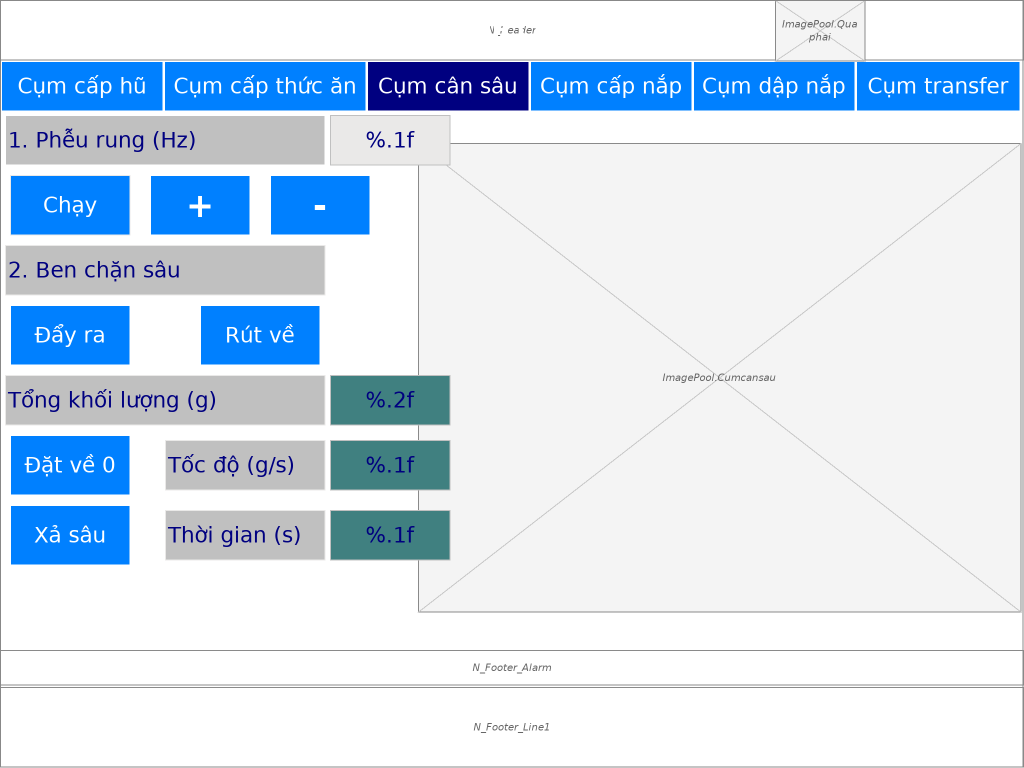
VISUALIZATION N_WormWeight1  // 1024x768
    Image (418,143 603x469), image: ImagePool.Cumcansau
    Rectangle (10,175 120x60), "Dừng", invisible if: not PR_Line01.bMotor_vibrating_funnel, input disabled if: not PR_Line01.bMotor_vibrating_funnel
        OnMouseDown: execute { PR_Line01.bMotor_vibrating_funnel := FALSE; PR_Line01.bxa := FALSE; }
    Rectangle (10,175 120x60), "Chạy", invisible if: PR_Line01.bMotor_vibrating_funnel, input disabled if: PR_Line01.bMotor_vibrating_funnel
        OnMouseDown: execute { PR_Line01.bMotor_vibrating_funnel := TRUE; PR_Line01.bxa := FALSE; }
    Rectangle (10,305 120x60), "Đẩy ra", colour toggle: PR_Line01.bCylinder_Block_Worm_Extend
        OnMouseDown: execute {
            PR_Line01.bCylinder_Block_Worm_Extend := TRUE;
            PR_Line01.bCylinder_Block_Worm_Retract := FALSE;
            PR_Line01.bxa := FALSE;
        }
    Rectangle (200,305 120x60), "Rút về", colour toggle: PR_Line01.bCylinder_Block_Worm_Retract
        OnMouseDown: execute {
            PR_Line01.bCylinder_Block_Worm_Retract := TRUE;
            PR_Line01.bCylinder_Block_Worm_Extend := FALSE;
            PR_Line01.bxa := FALSE;
        }
    Frame (0,687 1024x80)
        shows N_Footer_Line1()
    Frame (0,0 1024x60)
        shows N_Header()
    Textfield (353,5 400x50), "MÀN HÌNH CHẠY TAY LINE 1"
    Rectangle (5,115 320x50), "1. Phễu rung (Hz)"
    Rectangle (5,245 320x50), "2. Ben chặn sâu"
    Rectangle (1,61 162x50), "Cụm cấp hũ"
        OnMouseClick: change screen: N_JarSupply1
    Rectangle (164,61 202x50), "Cụm cấp thức ăn"
        OnMouseClick: change screen: N_FoodSupply1
    Rectangle (367,61 162x50), "Cụm cân sâu"
        OnMouseClick: change screen: N_WormWeight1
    Rectangle (530,61 162x50), "Cụm cấp nắp"
        OnMouseClick: change screen: N_LidSupply1
    Rectangle (693,61 162x50), "Cụm dập nắp"
        OnMouseClick: change screen: N_LidPressing1
    Rectangle (856,61 164x50), "Cụm transfer"
        OnMouseClick: change screen: N_Tranfer1
    Rectangle (330,115 120x50), "%.1f", text variable: PR_Line01.fb_WormWeight.fSpeed_vibrating_funnel_Manual
        OnMouseDown: write PR_Line01.fb_WormWeight.fSpeed_vibrating_funnel_Manual via VisuDialogs.Numpad
        OnMouseDown: execute { PR_Line01.bxa := FALSE; }
    Rectangle (5,375 320x50), "Tổng khối lượng (g)"
    Rectangle (150,175 100x60), "+", colour toggle: PR_Line01.bUp_vibrating_funnel
        OnMouseDown: execute { PR_Line01.bUp_vibrating_funnel := TRUE; PR_Line01.bxa := FALSE; }
    Rectangle (270,175 100x60), "-", colour toggle: PR_Line01.bDown_vibrating_funnel
        OnMouseDown: execute { PR_Line01.bDown_vibrating_funnel := TRUE; PR_Line01.bxa := FALSE; }
    Rectangle (330,375 120x50), "%.2f", text variable: PR_Line01.fb_WormWeight.fWeight_Worm
    Rectangle (10,435 120x60), "Đặt về 0"
        tap PR_Line01.bZero_Loadcell_Worm
        OnMouseDown: execute { PR_Line01.bxa := FALSE; }
        OnMouseUp: execute { PR_Line01.bZero_Loadcell_Worm := TRUE; }
    Rectangle (165,440 160x50), "Tốc độ (g/s)"
    Rectangle (330,440 120x50), "%.1f", text variable: PR_Line01.fb_WormWeight.fFlow_Worm
    Image (775,0 90x61), input disabled if: bResetAuto2, image: ImagePool.Qua phai
        OnMouseClick: change screen: N_WormWeight2
        OnMouseClick: execute { MAIN_LINE2.bModeManual := TRUE; MAIN_LINE2.bModeAuto := FALSE; }
    Rectangle (10,505 120x60), "Xả sâu", colour toggle: PR_Line01.xasau
        OnMouseDown: execute { PR_Line01.xasau := TRUE; PR_Line01.bxa := true; }
    Rectangle (165,510 160x50), "Thời gian (s)"
    Rectangle (330,510 120x50), "%.1f", text variable: PR_Line01.fb_WormWeight.fTime
    Frame (0,650 1024x35)
        shows N_Footer_Alarm()
END_VISUALIZATION

(* stored: Version 1.1.0.1, ProductVersion 3.1.4024.12
   Visu N_WormWeight1: Id {d9506cab-4aeb-4e38-b4c1-b9b4789c20a5} *)
